// TIA Portal project "Pumpensicherung_FUP" (V16)

(* hardware
DEVICE "S71500/ET200MP station_1"  S7-1500 station
   slot 0: "Rail_0"  Rack  6ES7 590-1***0-0AA0
   slot 1: "PLC_1"  CPU 1511-1 PN  6ES7 511-1AK00-0AB0  V1.8
      slot 3: "CPU display_1"  6ES7591-1AA00-0AA0
      slot 32768: "PROFINET interface_1"  X1
         slot 32769: "Port_1"  X1 P1
         slot 32770: "Port_2"  X1 P2
   slot 2: "DI 16x24VDC BA_1"  DI 16x24VDC BA  6ES7 521-1BH10-0AA0  V1.1
   slot 3: "DQ 8x24VDC/2A HF_1"  DQ 8x24VDC/2A HF  6ES7 522-1BF00-0AB0  V2.2
   slot 4: "AI 4xU/I/RTD/TC ST_1"  AI 4xU/I/RTD/TC ST  6ES7 531-7QD00-0AB0  V1.0
*)

// ===== PLC "PLC_1"  CPU 1511-1 PN =====

VAR_GLOBAL   // PLC tag table "Default tag table"
   "Strömungsschalter" AT %I0.0 : Bool;
   "Alarm-Reset" AT %I0.1 : Bool;
   "Alarmstummschalter" AT %I0.2 : Bool;
   "Hand-taste" AT %I0.3 : Bool;
   "Aus-Taste" AT %I0.4 : Bool;
   "Auto-Taste" AT %I0.5 : Bool;
   "Pumpe" AT %Q0.0 : Bool;
   "Strömungsschalterdefektleuchte" AT %Q0.1 : Bool;
   "Drucksensordefektleuchte" AT %Q0.2 : Bool;
   "Strömungschalter_Bit" AT %M4.0 : Bool;
   "Alarm-Reset_Bit" AT %M4.1 : Bool;
   "Alarmstummschalter_Bit" AT %M4.2 : Bool;
   "Hand_Taste_Bit" AT %M4.3 : Bool;
   "Aus_Taste_Bit" AT %M4.4 : Bool;
   "Auto_Taste_Bit" AT %M4.5 : Bool;
   "HOA_Modi" AT %MW6 : Int;   // 0 = AUS ; 1 = HAND ; 2 = AUTO
   "ONS1" AT %M4.6 : Bool;
   "ONS2" AT %M4.7 : Bool;
   "ONS3" AT %M5.0 : Bool;
   "Modus_vor_Hand" AT %MW8 : Int;
   "ONS4" AT %M5.3 : Bool;
   "Pumpe_AUTO_MODUS" AT %MW10 : Int;   // 1 = AN ; 0 = AUS
   "Pumpe_Interrupt" AT %M5.4 : Bool;
   "Strömungsschalterdefektleuchte_Bit" AT %M5.5 : Bool;
   "Pumpe_Bit" AT %M5.6 : Bool;
   "Drucksensordefektleuchte_Bit" AT %M5.7 : Bool;
   "Strömungsstörung_Alarmmeldung_Bit" AT %M12.0 : Bool;
   "Überdrucklalarmmeldung_Bit" AT %M12.1 : Bool;
   "Drucksensor_Ersatz" AT %MW14 : Int;
   "Druck in PSI" AT %MD16 : Real;
   "Alarm_Bit" AT %M0.0 : Bool;
   "One Shot" AT %M0.1 : Bool;
END_VAR

DATA_BLOCK "IO_DB"   // DB5
{ S7_Optimized_Access := 'TRUE' }
VERSION : 0.1
// stored: InstanceOfName IO
"IO"
BEGIN
END_DATA_BLOCK

DATA_BLOCK "HOA_DB"   // DB6
{ S7_Optimized_Access := 'TRUE' }
VERSION : 0.1
// stored: InstanceOfName HOA
"HOA"
BEGIN
END_DATA_BLOCK

DATA_BLOCK "Steuerung_DB"   // DB7
{ S7_Optimized_Access := 'TRUE' }
VERSION : 0.1
// stored: InstanceOfName Steuerung
"Steuerung"
BEGIN
END_DATA_BLOCK

DATA_BLOCK "Alarms_DB"   // DB8
{ S7_Optimized_Access := 'TRUE' }
VERSION : 0.1
// stored: InstanceOfName Alarms
"Alarms"
BEGIN
END_DATA_BLOCK

// folder: System blocks/Program resources

DATA_BLOCK "Pumpe_Aus_Verzögerung"   // DB1
{ S7_Optimized_Access := 'TRUE' }
AUTHOR : Simatic
FAMILY : IEC
NAME : IEC_TMR
VERSION : 1.0
// stored: InstanceOfName IEC_TIMER
"IEC_TIMER"
BEGIN
END_DATA_BLOCK

DATA_BLOCK "Pumpe_An_Verzögerung"   // DB2
{ S7_Optimized_Access := 'TRUE' }
AUTHOR : Simatic
FAMILY : IEC
NAME : IEC_TMR
VERSION : 1.0
// stored: InstanceOfName IEC_TIMER
"IEC_TIMER"
BEGIN
END_DATA_BLOCK

DATA_BLOCK "Überdruckalarm"   // DB3
{ S7_Optimized_Access := 'TRUE' }
AUTHOR : Simatic
FAMILY : IEC
NAME : IEC_TMR
VERSION : 1.0
// stored: InstanceOfName IEC_TIMER
"IEC_TIMER"
BEGIN
END_DATA_BLOCK

DATA_BLOCK "Strömungsstörungalarm"   // DB4
{ S7_Optimized_Access := 'TRUE' }
AUTHOR : Simatic
FAMILY : IEC
NAME : IEC_TMR
VERSION : 1.0
// stored: InstanceOfName IEC_TIMER
"IEC_TIMER"
BEGIN
END_DATA_BLOCK

// folder: (top level)

FUNCTION_BLOCK "IO"   // FB1, FBD
{ S7_Optimized_Access := 'TRUE' }
VERSION : 0.1
   VAR
      "Normalisierter Wert" : Real;
   END_VAR
BEGIN

REGION Network 1
   // Eingänge
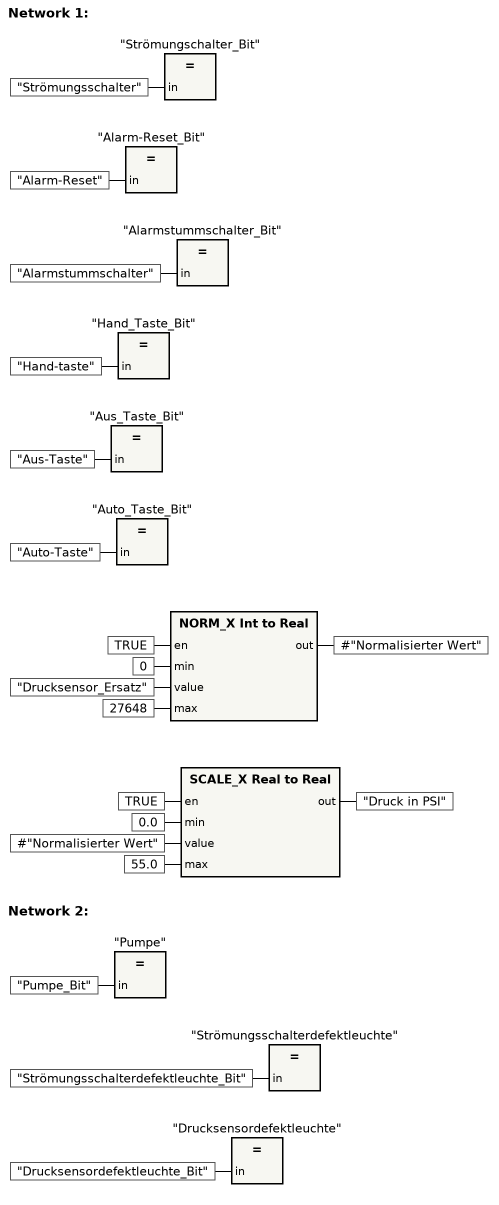
   "Strömungschalter_Bit" := "Strömungsschalter";
   "Alarm-Reset_Bit" := "Alarm-Reset";
   "Alarmstummschalter_Bit" := "Alarmstummschalter";
   "Hand_Taste_Bit" := "Hand-taste";
   "Aus_Taste_Bit" := "Aus-Taste";
   "Auto_Taste_Bit" := "Auto-Taste";
   IF TRUE THEN
       #"Normalisierter Wert" := NORM_X(MIN := 0, VALUE := "Drucksensor_Ersatz", MAX := 27648);
       "Druck in PSI" := SCALE_X(MIN := 0.0, VALUE := #"Normalisierter Wert", MAX := 55.0);
   END_IF;
END_REGION

REGION Network 2
   // Ausgänge
   "Pumpe" := "Pumpe_Bit";
   "Strömungsschalterdefektleuchte" := "Strömungsschalterdefektleuchte_Bit";
   "Drucksensordefektleuchte" := "Drucksensordefektleuchte_Bit";
END_REGION
END_FUNCTION_BLOCK

FUNCTION_BLOCK "Steuerung"   // FB2, FBD
{ S7_Optimized_Access := 'TRUE' }
VERSION : 0.1
   VAR
      Pumpe_Auto_Trigger : Bool;
      ONS_Auto : Bool;
      Pumpe_AUTO_Bit : Bool;
      ONS_HAND : Bool;
      Pumpe_Hand_Trigger : Bool;
      Pumpe_HAND_Bit : Bool;
      ONS_Strömung : Bool;
      ONS_Druck : Bool;
      ONS_Reset : Bool;
   END_VAR
   VAR_TEMP   // added for the SCL form of the ladder/FBD networks
      _w1 : Bool;
      _w2 : Bool;
      _w3 : Bool;
      _w4 : Bool;
   END_VAR
BEGIN

REGION Network 1
   // AUTO Steuerung
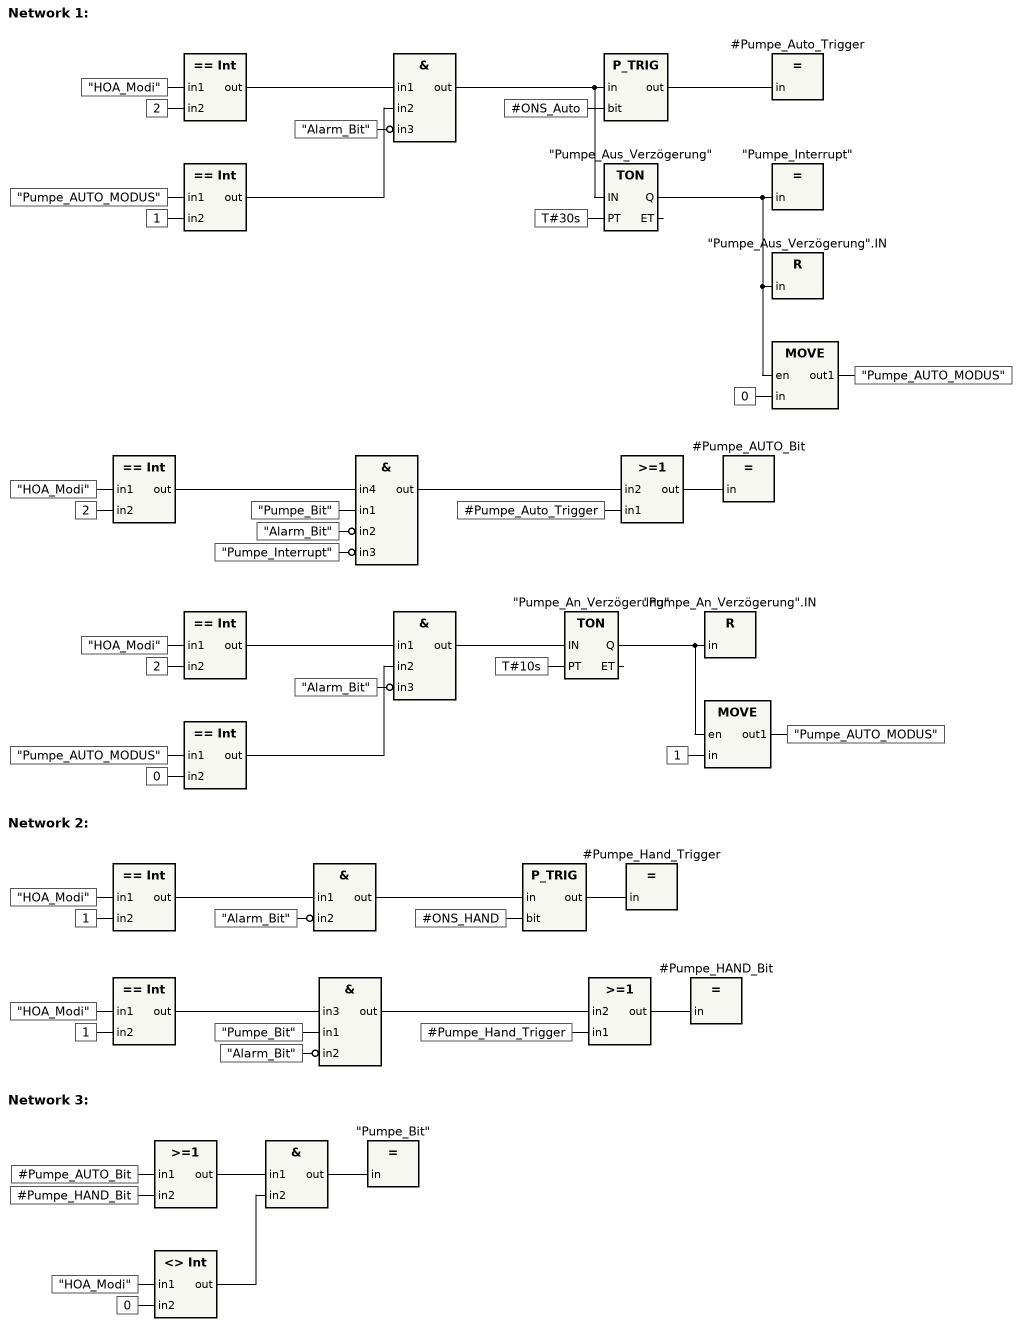
   #_w1 := ("HOA_Modi" = 2) AND ("Pumpe_AUTO_MODUS" = 1) AND NOT "Alarm_Bit";
   #_w2 := #_w1 AND NOT #ONS_Auto;   // rising edge
   #ONS_Auto := #_w1;
   #Pumpe_Auto_Trigger := #_w2;
   "Pumpe_Aus_Verzögerung".TON(IN := #_w1, PT := T#30s);
   "Pumpe_Interrupt" := "Pumpe_Aus_Verzögerung".Q;
   #_w3 := "Pumpe_Aus_Verzögerung".Q;
   IF #_w3 THEN
       "Pumpe_Aus_Verzögerung".IN := FALSE;
       "Pumpe_AUTO_MODUS" := 0;
   END_IF;
   #Pumpe_AUTO_Bit := (("HOA_Modi" = 2) AND "Pumpe_Bit" AND NOT "Alarm_Bit" AND NOT "Pumpe_Interrupt") OR #Pumpe_Auto_Trigger;
   "Pumpe_An_Verzögerung".TON(IN := ("HOA_Modi" = 2) AND ("Pumpe_AUTO_MODUS" = 0) AND NOT "Alarm_Bit",
                           PT := T#10s);
   #_w4 := "Pumpe_An_Verzögerung".Q;
   IF #_w4 THEN
       "Pumpe_An_Verzögerung".IN := FALSE;
       "Pumpe_AUTO_MODUS" := 1;
   END_IF;
END_REGION

REGION Network 2
   // HAND Steuerung
   #_w1 := ("HOA_Modi" = 1) AND NOT "Alarm_Bit";
   #_w2 := #_w1 AND NOT #ONS_HAND;   // rising edge
   #ONS_HAND := #_w1;
   #Pumpe_Hand_Trigger := #_w2;
   #Pumpe_HAND_Bit := (("HOA_Modi" = 1) AND "Pumpe_Bit" AND NOT "Alarm_Bit") OR #Pumpe_Hand_Trigger;
END_REGION

REGION Network 3
   // Pumpen_Steuerung
   "Pumpe_Bit" := (#Pumpe_AUTO_Bit OR #Pumpe_HAND_Bit) AND ("HOA_Modi" <> 0);
END_REGION

REGION Network 4
   // Alarm_Beleuchtung
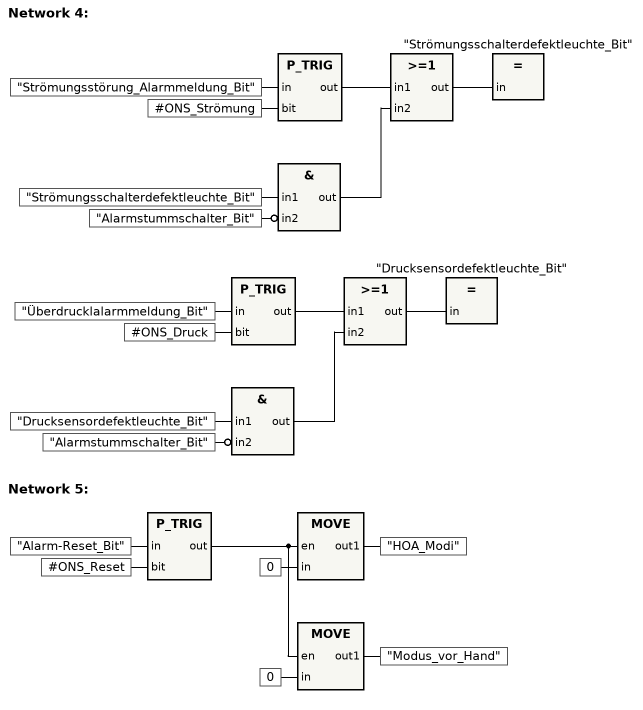
   #_w1 := "Strömungsstörung_Alarmmeldung_Bit" AND NOT #ONS_Strömung;   // rising edge
   #ONS_Strömung := "Strömungsstörung_Alarmmeldung_Bit";
   "Strömungsschalterdefektleuchte_Bit" := #_w1 OR ("Strömungsschalterdefektleuchte_Bit" AND NOT "Alarmstummschalter_Bit");
   #_w2 := "Überdrucklalarmmeldung_Bit" AND NOT #ONS_Druck;   // rising edge
   #ONS_Druck := "Überdrucklalarmmeldung_Bit";
   "Drucksensordefektleuchte_Bit" := #_w2 OR ("Drucksensordefektleuchte_Bit" AND NOT "Alarmstummschalter_Bit");
END_REGION

REGION Network 5
   // Alarm_Reset
   #_w1 := "Alarm-Reset_Bit" AND NOT #ONS_Reset;   // rising edge
   #ONS_Reset := "Alarm-Reset_Bit";
   IF #_w1 THEN
       "HOA_Modi" := 0;
       "Modus_vor_Hand" := 0;
   END_IF;
END_REGION
END_FUNCTION_BLOCK

FUNCTION_BLOCK "HOA"   // FB3, FBD
{ S7_Optimized_Access := 'TRUE' }
VERSION : 0.1
   VAR
      AUTO_ONS : Bool;
      "ONS 5" : Bool;
   END_VAR
   VAR_TEMP   // added for the SCL form of the ladder/FBD networks
      _w1 : Bool;
      _w2 : Bool;
      _w3 : Bool;
      _w4 : Bool;
   END_VAR
BEGIN

REGION Network 1
   // HOA Auto
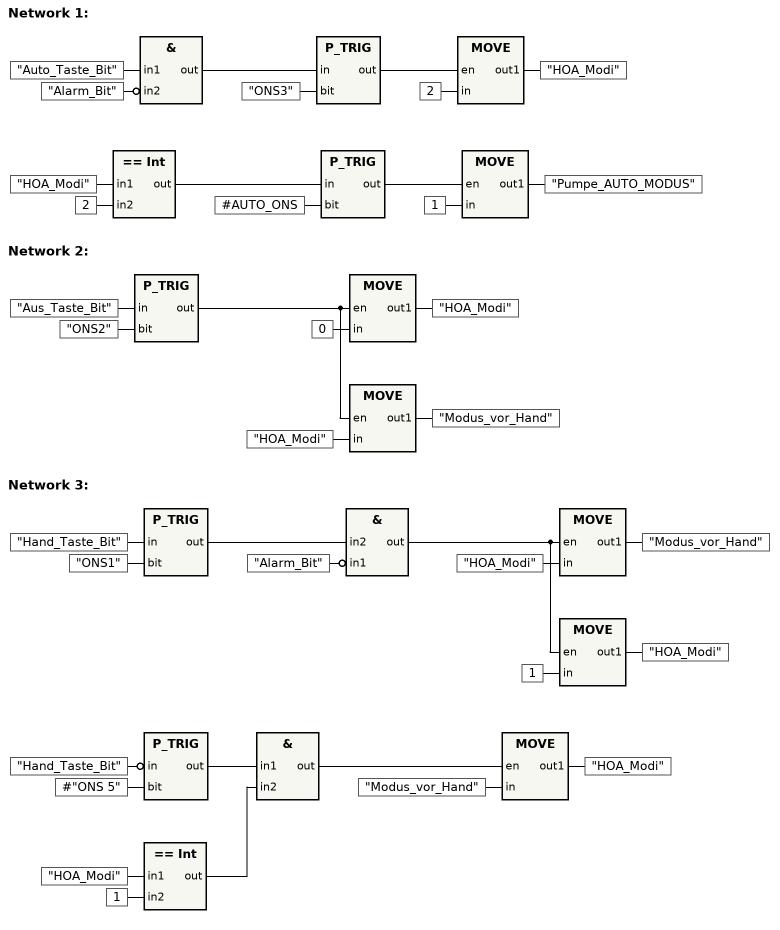
   #_w1 := "Auto_Taste_Bit" AND NOT "Alarm_Bit";
   #_w2 := #_w1 AND NOT "ONS3";   // rising edge
   "ONS3" := #_w1;
   IF #_w2 THEN "HOA_Modi" := 2; END_IF;
   #_w3 := "HOA_Modi" = 2;
   #_w4 := #_w3 AND NOT #AUTO_ONS;   // rising edge
   #AUTO_ONS := #_w3;
   IF #_w4 THEN "Pumpe_AUTO_MODUS" := 1; END_IF;
END_REGION

REGION Network 2
   // HOA Aus
   #_w1 := "Aus_Taste_Bit" AND NOT "ONS2";   // rising edge
   "ONS2" := "Aus_Taste_Bit";
   IF #_w1 THEN
       "HOA_Modi" := 0;
       "Modus_vor_Hand" := "HOA_Modi";
   END_IF;
END_REGION

REGION Network 3
   // HOA Hand
   #_w1 := "Hand_Taste_Bit" AND NOT "ONS1";   // rising edge
   "ONS1" := "Hand_Taste_Bit";
   IF #_w1 AND NOT "Alarm_Bit" THEN
       "Modus_vor_Hand" := "HOA_Modi";
       "HOA_Modi" := 1;
   END_IF;
   #_w2 := NOT "Hand_Taste_Bit" AND NOT #"ONS 5";   // rising edge
   #"ONS 5" := NOT "Hand_Taste_Bit";
   IF #_w2 AND ("HOA_Modi" = 1) THEN "HOA_Modi" := "Modus_vor_Hand"; END_IF;
END_REGION
END_FUNCTION_BLOCK

FUNCTION_BLOCK "Alarms"   // FB4, FBD
{ S7_Optimized_Access := 'TRUE' }
VERSION : 0.1
   VAR
      ONS7 : Bool;
      ONS8 : Bool;
      Überdruckalarm_Trigger : Bool;
      Überdruckalarmmeldung_Trigger : Bool;
      Überdruck_Alarm : Bool;
      Strömungsstörung_Alarm : Bool;
      Strömungsstörung_Alarm_Trigger : Bool;
      ONS5 : Bool;
      ONS6 : Bool;
      Strömungsstörung_Alarmmeldung_Trigger : Bool;
   END_VAR
   VAR_TEMP   // added for the SCL form of the ladder/FBD networks
      _w1 : Bool;
      _w2 : Bool;
   END_VAR
BEGIN

REGION Network 1
   // Druckalarm
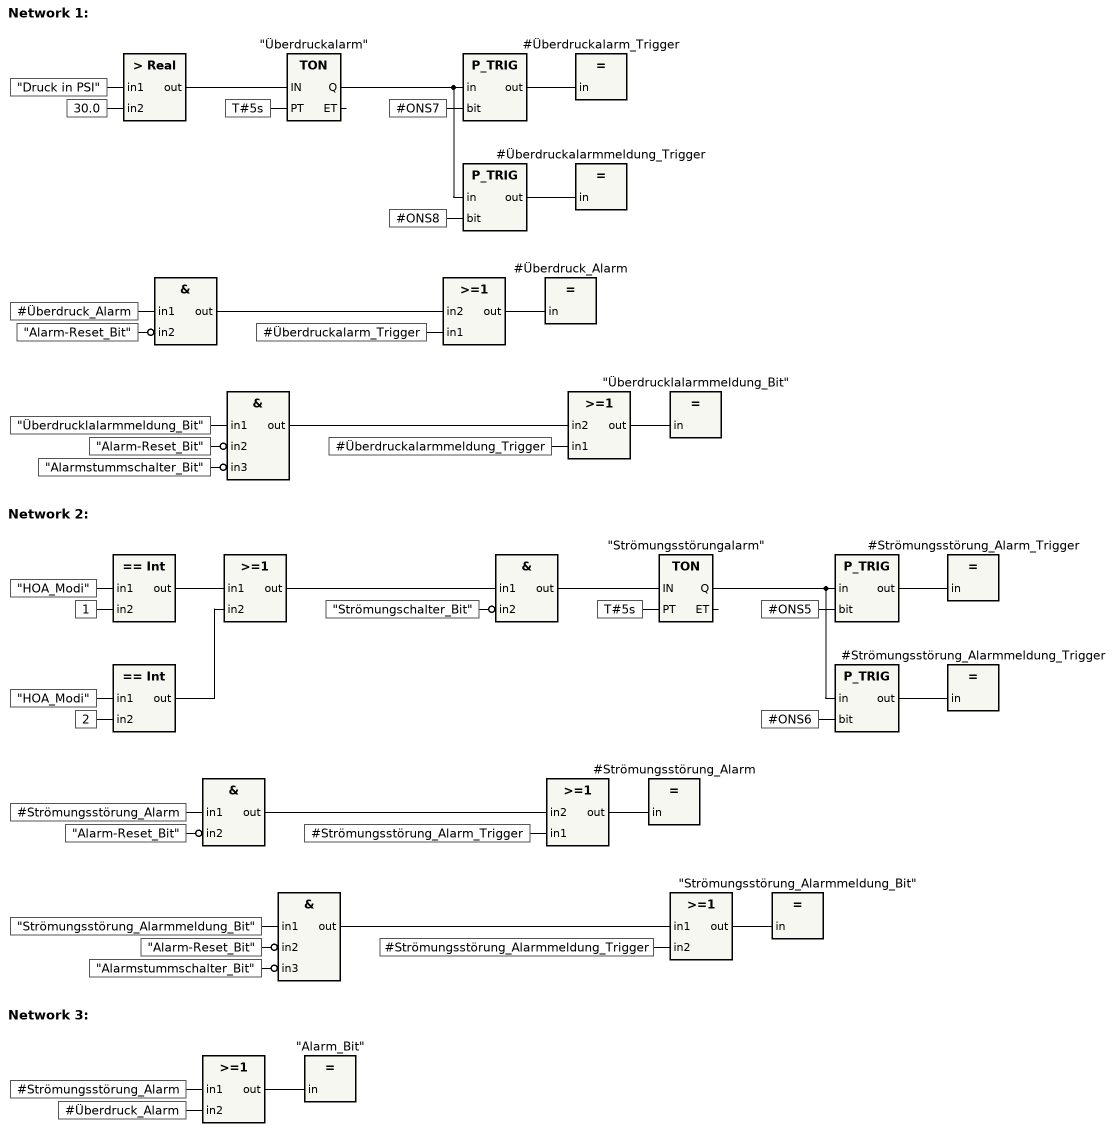
   "Überdruckalarm".TON(IN := "Druck in PSI" > 30.0, PT := T#5s);
   #_w1 := "Überdruckalarm".Q AND NOT #ONS7;   // rising edge
   #ONS7 := "Überdruckalarm".Q;
   #Überdruckalarm_Trigger := #_w1;
   #_w2 := "Überdruckalarm".Q AND NOT #ONS8;   // rising edge
   #ONS8 := "Überdruckalarm".Q;
   #Überdruckalarmmeldung_Trigger := #_w2;
   #Überdruck_Alarm := (#Überdruck_Alarm AND NOT "Alarm-Reset_Bit") OR #Überdruckalarm_Trigger;
   "Überdrucklalarmmeldung_Bit" := ("Überdrucklalarmmeldung_Bit" AND NOT "Alarm-Reset_Bit" AND NOT "Alarmstummschalter_Bit") OR #Überdruckalarmmeldung_Trigger;
END_REGION

REGION Network 2
   // Strömungsalarm
   "Strömungsstörungalarm".TON(IN := (("HOA_Modi" = 1) OR ("HOA_Modi" = 2)) AND NOT "Strömungschalter_Bit",
                           PT := T#5s);
   #_w1 := "Strömungsstörungalarm".Q AND NOT #ONS5;   // rising edge
   #ONS5 := "Strömungsstörungalarm".Q;
   #Strömungsstörung_Alarm_Trigger := #_w1;
   #_w2 := "Strömungsstörungalarm".Q AND NOT #ONS6;   // rising edge
   #ONS6 := "Strömungsstörungalarm".Q;
   #Strömungsstörung_Alarmmeldung_Trigger := #_w2;
   #Strömungsstörung_Alarm := (#Strömungsstörung_Alarm AND NOT "Alarm-Reset_Bit") OR #Strömungsstörung_Alarm_Trigger;
   "Strömungsstörung_Alarmmeldung_Bit" := ("Strömungsstörung_Alarmmeldung_Bit" AND NOT "Alarm-Reset_Bit" AND NOT "Alarmstummschalter_Bit") OR #Strömungsstörung_Alarmmeldung_Trigger;
END_REGION

REGION Network 3
   // Alarm_Bit
   "Alarm_Bit" := #Strömungsstörung_Alarm OR #Überdruck_Alarm;
END_REGION
END_FUNCTION_BLOCK

ORGANIZATION_BLOCK "Main"   // OB1, LAD, ProgramCycle
TITLE = "Main Program Sweep (Cycle)"
{ S7_Optimized_Access := 'TRUE' }
VERSION : 0.1
// PROJEKTBESCHREIBUNG: BEI DIESEM PROJEKT GEHT ES UM DIE SICHERHEIT DER PUMPE. DIE 
// SICHERHEIT DER PUMPE WIRD DURCH EINE KOMBINATION VON ZWEI SENSOREN GEWÄHRLEISTET:1) STRÖMUNGSSCHALTER 2) DRUCKSENSOR .DER STRÖMUNGSSCHALTER WIRD VOR DER PUMPE UND DER DRUCKSENSOR NACH DEM PUMPE MONTIERT. SOBALD DIE PUMPE AN IST UND FÜR FÜNF SEKUNDEN LÄUFT, WIRD ES FESTGESTELLT, OB DER STRÖMUNGSCHALTER GESCHLOSSEN IST UND/ODER OB DER DRUCK NACH DER PUMPE KLEINER ALS 30 PSI IST. WENN ES NICHT DER FALL IST, WIRD EIN ALARM AUSGELÖST UND DIE PUMPE AUSGESCHALTET. SOLANGE DANN DER ALARM-RESET NICHT BETÄTIGT WIRD, KANN DIE PUMPE NICHT WIEDER IM BETRIEB GENOMMEN WERDEN. AUßERDEM WIRD DIE PUMP MITTELS HAND/AUTOMATIK/AUS SCHALTER BETRIEBEN. SOLANGE DIE HANDTASTE GEDRUCKT BLEIBT, LÄUFT DIE PUMPE. SOBALD DIE HANDTASTE LOSGELASSEN WIRD GEHT DIE PUMPE WIRD IM MODUS, DAS VOR DEM HAND-MODUS AKTIV WAR. IN AUTO-MODUS LÄUFT DIE PUMPE IN EINEM ZYKLUS. DAS HEIßT, DIE PUMPE IST FÜR 30 SEKUNDEN AN UND DANN BLEIBT AUS FÜR 10 SEKUNDEN UND DANN WIEDER AN FÜR 30 SEKUNDEN UND SO WEITER. IM OFF-MODUS (AUS) BLEIBT DIE PUMPE AUS.
// 
// TESTKRITERIEN:
// 1) ZUNÄCHST BLEIBT DIE PUMPE AUS. SETZE DRUCKERSATZ AUF 13824 UND DER DRUCK SOLLTE 27,5 PSI BETRAGEN.
// 2) HANDTASTE WIRD GEDRUCKT BZW EINGESCHALTET. DIE PUMPE GEHT AN UND BLEIBT AN FÜR 5 SEKUNDEN UND DANN WIEDER AUS. DER ALARM WIRD AUSGELÖST UND DIE STRÖMUNGSSCHALTERDEFEKTLEUCHTE LEUCHTET.
// 3) HANDTASTE WIRD LOSGELASSEN UND DER ALARMSTUMMSCHALTER WIRD BETÄTIGT UND DIE LEUCHTE GEHT WIEDER AUS. HANDTASTE WIRD FÜR EINIGE SEKUNDEN GEDRUCKT UND WIEDER LOSGELASSEN ABER DIE PUMPE GEHT NICHT AN.
// 4) AUTOTASTE WIRD GETOGGELT. DIE PUMPEZYKLUS SOLLTE NICHT AN GEHEN
// 5) ALARMRESET WIRD BETÄTIGT UND DANN WIRD STRÖMUNGSCHALTER GESCHALTET. NUN WIRD AUTOTASTE GETOGGELT. DIE PUMPE SOLLTE IM ZYKLUS LAUFEN. 
// 6) NUN WIRD HANDTASTE GEDRUCKT FÜR UNGEFÄHR 20 SEKUNDEN. DIE PUMPE SOLLTE AUS DEM ZYKLUS RAUS UND STÄNDIG LAUFEN. WIRD DIE HANDTASTE WIEDER GELASSEN SOLLTE DIE PUMPE WIRD IM ZYKLUS LAUFEN.
// 7) SETZE DRUCKERSATZ AUF 16876 UND DIE PUMPE SOLLTE NACH 5 SEKUNDEN AUS GEHEN. DER ALARM WIRD AUSGELÖST UND DIE DRUCKSENSORDEFEKTLEUCHTE LEUCHTET. DER DRUCKWERT BETRÄGT 33,5 PSI.
   VAR_INPUT
      Initial_Call : Bool;   // Initial call of this OB
      Remanence : Bool;   // =True, if remanent data are available
   END_VAR
BEGIN

REGION Network 1
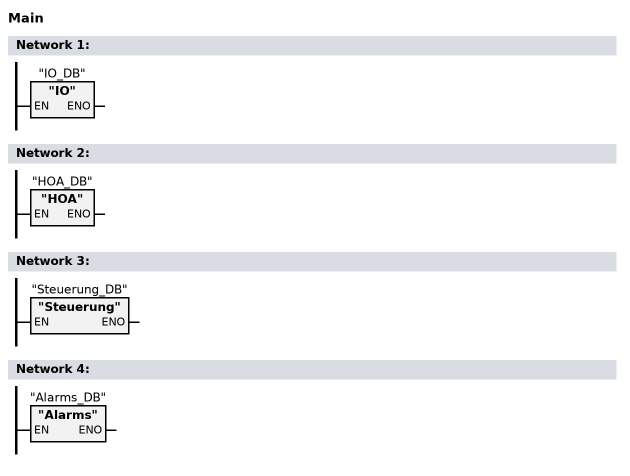
   RUNG wire#powerrail
      "IO_DB"()
   END_RUNG
   // the same network as SCL:
   "IO_DB"();   // "IO"
END_REGION

REGION Network 2
   RUNG wire#powerrail
      "HOA_DB"()
   END_RUNG
   // the same network as SCL:
   "HOA_DB"();   // "HOA"
END_REGION

REGION Network 3
   RUNG wire#powerrail
      "Steuerung_DB"()
   END_RUNG
   // the same network as SCL:
   "Steuerung_DB"();   // "Steuerung"
END_REGION

REGION Network 4
   RUNG wire#powerrail
      "Alarms_DB"()
   END_RUNG
   // the same network as SCL:
   "Alarms_DB"();   // "Alarms"
END_REGION
END_ORGANIZATION_BLOCK